PROGRAM MAIN
VAR
	machine_level_piper : Piper();
	task_fb : TaskFB();
	piper_em : Piper_EM(machine_level_piper, task_fb);
END_VAR

machine_level_piper();
task_fb();
piper_em();

END_PROGRAM

(* stored: Version 1.1.0.1, ProductVersion 3.1.4024.12
   POU MAIN: Id {a3a46004-2020-4778-9fbf-7f2bc7484f47}, SpecialFunc None *)
